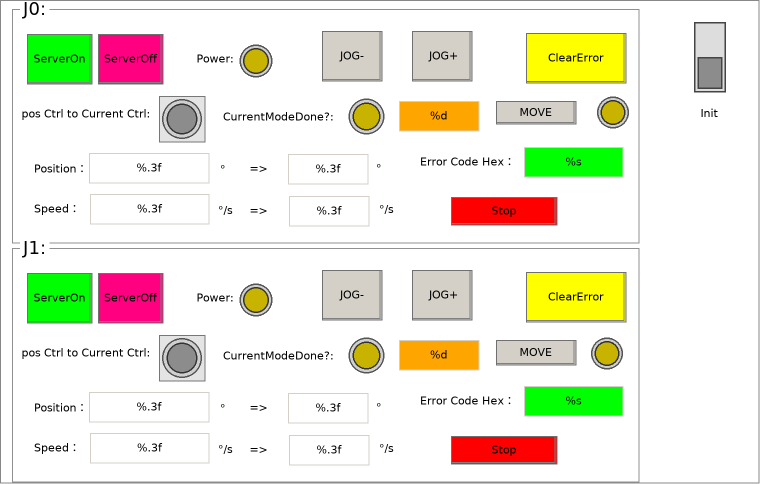
VISUALIZATION StatJoint  // 760x484
    GroupBox (12,1 627x242), "J0:"
        Textfield (77,152 120x30), "%.3f", text variable: MAIN.AxisInfo[0].PositionCmd
        Label (6,94 136x38), "pos Ctrl to Current Ctrl:"
        Label (198,154 22x29), "°"
        Label (13,192 64x32), "Speed："
        Textfield (78,193 119x30), "%.3f", text variable: MAIN.AxisMotionPara[0].TargetVelocity
            OnMouseClick: write the text variable via VisuDialogs.Numpad
        Label (193,195 37x29), "°/s"
        Button (86,33 65x50), "ServerOff", input disabled if: NOT MAIN.AxisOp[0].AxisInfo.AxisStatus.Ready
            toggle MAIN.HMI_AxisEnable[0]
        Button (514,32 100x50), "ClearError"
            tap MAIN.HMI_Axis_reset[0]
        Label (173,43 60x30), "Power:"
        Label (261,47 40x30)
        Button (310,30 60x50), "JOG-"
            tap MAIN.HMI_AxisJogBackwards[0]
        Button (400,30 60x50), "JOG+"
            tap MAIN.HMI_AxisJogFoward[0]
        Textfield (276,153 80x30), "%.3f", text variable: MAIN.AxisInfo[0].ActualPosition
        Label (354,153 22x29), "°"
        Label (354,194 37x29), "°/s"
        Textfield (277,195 80x30), "%.3f", text variable: MAIN.AxisInfo[0].ActualVelocity
        Textfield (387,100 80x30), "%d", text variable: MAIN.HMI_TargetTorque[0]
            OnMouseClick: write the text variable via VisuDialogs.Numpad
        Label (406,146 99x30), "Error Code Hex："
        Textfield (512,146 99x30), "%s", text variable: MAIN.AxisOp[0].AxisInfo.ErrId_Hex
        Label (224,149 45x38), "=>"
        Label (224,191 45x38), "=>"
        Button (15,33 65x50), "ServerOn", input disabled if: NOT MAIN.AxisOp[0].AxisInfo.AxisStatus.Ready
            toggle MAIN.HMI_AxisEnable[0]
        PushSwitchLed (146,95 48x46), variable: MAIN.HMI_CurrentControlOfEnable[0], behaviour: TOGGLE, style: Switch-PushSwitchLed-Gray
        Label (18,149 62x38), "Position："
        Button (439,196 106x28), "Stop"
            tap MAIN.HMI_AxisStop[0]
        Lamp1 (225,40 38x40), variable: MAIN.AxisOp[0].AxisInfo.AxisStatus.Enabled, style: Lamp-Lamp1-Yellow
        Label (209,97 115x38), "CurrentModeDone?:"
        Lamp1 (334,94 41x43), variable: MAIN.HMI_AxisCurrentControlFlag[0], style: Lamp-Lamp1-Yellow
        Button (484,100 80x23), "MOVE"
            toggle MAIN.HMI_CurrentControlMove[0]
    DipSwitch (675,22 70x70), variable: MAIN.SiasunServoTestStart, behaviour: TOGGLE, style: Switch-DipSwitch-Gray
    Label (661,100 97x27), "Init"
    GroupBox (12,240 627x242), "J1:"
        Textfield (77,152 120x30), "%.3f", text variable: MAIN.AxisInfo[1].PositionCmd
        Label (6,94 136x38), "pos Ctrl to Current Ctrl:"
        Label (198,154 22x29), "°"
        Label (13,192 64x32), "Speed："
        Textfield (78,193 119x30), "%.3f", text variable: MAIN.AxisMotionPara[1].TargetVelocity
            OnMouseClick: write the text variable via VisuDialogs.Numpad
        Label (193,195 37x29), "°/s"
        Button (86,33 65x50), "ServerOff", input disabled if: NOT MAIN.AxisOp[1].AxisInfo.AxisStatus.Ready
            toggle MAIN.HMI_AxisEnable[1]
        Button (514,32 100x50), "ClearError"
            tap MAIN.HMI_Axis_reset[1]
        Label (173,43 60x30), "Power:"
        Label (261,47 40x30)
        Button (310,30 60x50), "JOG-"
            tap MAIN.HMI_AxisJogBackwards[1]
        Button (400,30 60x50), "JOG+"
            tap MAIN.HMI_AxisJogFoward[1]
        Textfield (276,153 80x30), "%.3f", text variable: MAIN.AxisInfo[1].ActualPosition
        Label (354,153 22x29), "°"
        Label (354,194 37x29), "°/s"
        Textfield (277,195 80x30), "%.3f", text variable: MAIN.AxisInfo[1].ActualVelocity
        Textfield (387,100 80x30), "%d", text variable: MAIN.HMI_TargetTorque[1]
            OnMouseClick: write the text variable via VisuDialogs.Numpad
        Button (484,100 80x25), "MOVE"
            toggle MAIN.HMI_CurrentControlMove[1]
        Label (406,146 99x30), "Error Code Hex："
        Textfield (512,146 99x30), "%s", text variable: MAIN.AxisOp[1].AxisInfo.ErrId_Hex
        Label (224,149 45x38), "=>"
        Label (224,191 45x38), "=>"
        Button (15,33 65x50), "ServerOn", input disabled if: NOT MAIN.AxisOp[1].AxisInfo.AxisStatus.Ready
            toggle MAIN.HMI_AxisEnable[1]
        PushSwitchLed (146,95 48x46), variable: MAIN.HMI_CurrentControlOfEnable[1], behaviour: TOGGLE, style: Switch-PushSwitchLed-Gray
        Label (18,149 62x38), "Position："
        Button (439,196 106x28), "Stop"
            tap MAIN.HMI_AxisStop[1]
        Lamp1 (225,40 38x40), variable: MAIN.AxisOp[1].AxisInfo.AxisStatus.Enabled, style: Lamp-Lamp1-Yellow
        Label (209,97 115x38), "CurrentModeDone?:"
        Lamp1 (334,94 41x43), variable: MAIN.HMI_AxisCurrentControlFlag[1], style: Lamp-Lamp1-Yellow
        Lamp1 (575,95 40x37), variable: MAIN.HMI_CurrentControlMove[1], style: Lamp-Lamp1-Yellow
    Lamp1 (593,94 40x37), variable: MAIN.HMI_CurrentControlMove[0], style: Lamp-Lamp1-Yellow
END_VISUALIZATION

(* stored: Version 1.1.0.1, ProductVersion 3.1.4024.12
   Visu StatJoint: Id {38e30f9e-af14-4b84-aac3-ba341e33396b} *)
